KUKA KRL data list: test.dat

&ACCESS RVO
DEFDAT test
;FOLD EXTERNAL DECLARATIONS;%{PE}%MKUKATPBASIS,%CEXT,%VCOMMON,%P
  ;FOLD BASISTECH EXT;%{PE}%MKUKATPBASIS,%CEXT,%VEXT,%P
    EXT  BAS (BAS_COMMAND  :IN,REAL  :IN )
  ;ENDFOLD (BASISTECH EXT)

  EXT sPlanen2()
  EXT sTasche1()
  EXT sParallel2()
  EXT sKontur5()

;ENDFOLD (EXTERNAL DECLARATIONS)
ENDDAT
